TYPE ST_HMI_MANUAL_DEVICE_IN :
STRUCT
	stButtonOn,
	stButtonOff	: ST_HMI_BUTTON_IN;
	
	fValue		: REAL;
END_STRUCT
END_TYPE

(* stored: Version 1.1.0.1
   DUT ST_HMI_MANUAL_DEVICE_IN: Id {a4f79744-f573-40d6-8741-9318db7d300a} *)
